// TIA Portal V20 export
DATA_BLOCK "DB_NordSetPoint"   // DB33
// stored: Access Published, MemoryReserve 100, Namespace Global
   VAR
      Line : Struct
         A1 : Struct   // -(0 - 16000) -> (CW: 0 - 100%) || +(0 - 16000) (CCW: 0 - 100%) || freq. has been set via NORDCON
            Conveyor : Array[_.gMinA1.._.gMaxA1] of DInt;
         END_STRUCT;
         B1 : Struct   // -(0 - 16000) -> (CW: 0 - 100%) || +(0 - 16000) (CCW: 0 - 100%) || freq. has been set via NORDCON
            Conveyor : Array[_.gMinB1.._.gMaxB1] of DInt;
         END_STRUCT;
         C1 : Struct   // -(0 - 16000) -> (CW: 0 - 100%) || +(0 - 16000) (CCW: 0 - 100%) || freq. has been set via NORDCON
            Conveyor : Array[_.gMinC1.._.gMaxC1] of DInt;
         END_STRUCT;
         D1 : Struct   // -(0 - 16000) -> (CW: 0 - 100%) || +(0 - 16000) (CCW: 0 - 100%) || freq. has been set via NORDCON
            Conveyor : Array[_.gMinD1.._.gMaxD1] of DInt;
         END_STRUCT;
      END_STRUCT;
   END_VAR
BEGIN
END_DATA_BLOCK
